//==================================================================================================
//							Beckhoff Automation Poland
//									03.01.2023
//
// Code owner: TG
//
// Sample code to maitenance software limit switches
//
// Used libraries: 
//	Tc2_MC2							|| 3.3.48.0
//	Tc2_System						|| 3.4.26.0
//
//
// 	v2.0 	|| TC v 3.1.4024.35 	|| Second edition - OOP based
// 	v1.0 	|| TC v 3.1.4020.32 	|| First edition
//==================================================================================================
{attribute 'reflection'}
FUNCTION_BLOCK FB_NcSWLimitSwitchCtrlv2
VAR CONSTANT
	udiIDXGRP_OFFS								: UDINT := 16#0000_5000;
END_VAR
VAR
	{attribute 'instance-path'}
	{attribute 'noinit'}
	sInstancePath								: STRING;

	_stRead										: Tc2_MC2.ST_McOutputs;
	_stWrite									: Tc2_MC2.ST_McOutputs;
	_lrLimitSwitchPositionMin					: LREAL 		:= 0;
	_lrLimitSwitchPositionMax					: LREAL 		:= 0;
	_bLimitSwitchStateMin						: BOOL 			:= FALSE;
	_bLimitSwitchStateMax						: BOOL 			:= FALSE;
	bAxisIdError								: BOOL;
END_VAR

PROPERTY LimitSwitchPositionMax 				: LREAL
GET
LimitSwitchPositionMax							:= _lrLimitSwitchPositionMax;
END_GET
SET
_lrLimitSwitchPositionMax						:= LimitSwitchPositionMax;
END_SET
END_PROPERTY

PROPERTY LimitSwitchPositionMin 				: LREAL
GET
LimitSwitchPositionMin							:= _lrLimitSwitchPositionMin;
END_GET
SET
_lrLimitSwitchPositionMin						:= LimitSwitchPositionMin;
END_SET
END_PROPERTY

PROPERTY LimitSwitchStateMax 					: BOOL
GET
LimitSwitchStateMax								:= _bLimitSwitchStateMax;
END_GET
SET
_bLimitSwitchStateMax							:= LimitSwitchStateMax;
END_SET
END_PROPERTY

PROPERTY LimitSwitchStateMin 					: BOOL
GET
LimitSwitchStateMin							:= _bLimitSwitchStateMin;
END_GET
SET
_bLimitSwitchStateMin							:= LimitSwitchStateMin;
END_SET
END_PROPERTY

PROPERTY pRead 							: Tc2_MC2.ST_McOutputs
GET
pRead											:= _stRead;
END_GET
SET
_stRead											:= pRead;
END_SET
END_PROPERTY

PROPERTY pWrite 							: Tc2_MC2.ST_McOutputs
GET
pWrite											:= _stWrite;
END_GET
SET
_stWrite										:= pWrite;
END_SET
END_PROPERTY

// Needs one cycle extra with false execution, after busy false
METHOD ReadBool 								: Tc2_MC2.ST_McOutputs
VAR_INPUT
	bExecute									: BOOL;
	nAxisID										: UDINT;
	nOffset										: UDINT;
END_VAR
VAR_OUTPUT
	bOut										: BOOL;
END_VAR
VAR_INST
	fbADSREAD									: ADSREAD;
	wData										: WORD;
	nStep										: DINT;
END_VAR
VAR
	Out											: Tc2_MC2.ST_McOutputs;
	Message										: STRING;
END_VAR
IF nAxisID = 0 THEN
	
	IF NOT bAxisIdError THEN
		ADSLOGSTR(ADSLOG_MSGTYPE_ERROR,'FB_NcSWLimitSwitchCtrl critical error - Axis ID not assigned! FB instance: %s',sInstancePath);
	END_IF
	
	bAxisIdError 								:= TRUE;
	RETURN;	
END_IF

fbADSREAD(			PORT						:= 500, 
					IDXGRP						:= udiIDXGRP_OFFS + nAxisID, 
					IDXOFFS						:= nOffset, 
					LEN							:= 2, 
					DESTADDR					:= ADR(wData), 
					READ						:= bExecute, 
					BUSY						=> Out.Busy, 
					ERR							=> Out.Error, 
					ERRID						=> Out.ErrorID);

// Fix library issue, one extra cycle + Done
CASE nStep OF
	
	0: 
	
		Out.Error 								:= FALSE;
		Out.ErrorID 							:= 0;

		IF Out.Busy THEN
			nStep								:= nStep + 10;
		END_IF
	
	10:
	
		IF NOT Out.Busy THEN
			Out.Busy							:= TRUE;
			IF Out.Error THEN
				Out.ErrorID						:= 0;
				Out.Error						:= FALSE;
				nStep							:= 1000;
			ELSE
				nStep							:= 100;
			END_IF
		END_IF
		
	100, 1000:

		Out.Done								:= nStep = 100;
		Out.Error								:= nStep = 1000;
		IF Out.Error THEN
			Message := CONCAT('FB_NcSWLimitSwitchCtrl method ReadBool failed - Error ID: ',UDINT_TO_STRING(Out.ErrorID));
			Message := CONCAT(Message, '! FB instance: %s');
			ADSLOGSTR(ADSLOG_MSGTYPE_WARN,Message,sInstancePath);
		END_IF
		
		IF bExecute THEN
			nStep								:= nStep + 1;
		ELSE
			fbADSREAD(	READ					:= FALSE);
			nStep								:= 0;
		END_IF
		
	101, 1001:
	
		Out.Done								:= nStep = 101;
		Out.Error								:= nStep = 1001;
		IF NOT bExecute THEN
			fbADSREAD(	READ					:= FALSE);
			Out.Done							:= FALSE;
			Out.Error							:= FALSE;
			Out.ErrorID							:= 0;
			nStep								:= 0;
		END_IF	

END_CASE

pRead											:= Out;

bOut											:= wData.0;
ReadBool										:= Out;
END_METHOD

METHOD ReadLreal 								: Tc2_MC2.ST_McOutputs
VAR_INPUT
	bExecute									: BOOL;
	nAxisID										: UDINT;
	nOffset										: UDINT;
END_VAR
VAR_OUTPUT
	lrOut										: LREAL;
END_VAR
VAR_INST
	fbADSREAD									: ADSREAD;
	lrData										: LREAL;
	nStep										: DINT;
END_VAR
VAR
	Out											: Tc2_MC2.ST_McOutputs;
	Message										: STRING;
END_VAR
IF nAxisID = 0 THEN
	
	IF NOT bAxisIdError THEN
		ADSLOGSTR(ADSLOG_MSGTYPE_ERROR,'FB_NcSWLimitSwitchCtrl critical error - Axis ID not assigned! FB instance: %s',sInstancePath);
	END_IF
	
	bAxisIdError 								:= TRUE;
	RETURN;	
END_IF

fbADSREAD(			PORT						:= 500, 
					IDXGRP						:= udiIDXGRP_OFFS + nAxisID, 
					IDXOFFS						:= nOffset, 
					LEN							:= 8, 
					DESTADDR					:= ADR(lrData), 
					READ						:= bExecute, 
					BUSY						=> Out.Busy, 
					ERR							=> Out.Error, 
					ERRID						=> Out.ErrorID);

// Fix library issue, one extra cycle + Done
CASE nStep OF
	
	0: 
	
		Out.Error 								:= FALSE;
		Out.ErrorID 							:= 0;

		IF Out.Busy THEN
			nStep								:= nStep + 10;
		END_IF
	
	10:
	
		IF NOT Out.Busy THEN
			Out.Busy							:= TRUE;
			IF Out.Error THEN
				Out.ErrorID						:= 0;
				Out.Error						:= FALSE;
				nStep							:= 1000;
			ELSE
				nStep							:= 100;
			END_IF
		END_IF
		
	100, 1000:

		Out.Done								:= nStep = 100;
		Out.Error								:= nStep = 1000;
		IF Out.Error THEN
			Message := CONCAT('FB_NcSWLimitSwitchCtrl method ReadLreal failed - Error ID: ',UDINT_TO_STRING(Out.ErrorID));
			Message := CONCAT(Message, '! FB instance: %s');
			ADSLOGSTR(ADSLOG_MSGTYPE_WARN,Message,sInstancePath);
		END_IF
		
		IF bExecute THEN
			nStep								:= nStep + 1;
		ELSE
			fbADSREAD(	READ					:= FALSE);
			nStep								:= 0;
		END_IF
		
	101, 1001:
	
		Out.Done								:= nStep = 101;
		Out.Error								:= nStep = 1001;
		IF NOT bExecute THEN
			fbADSREAD(	READ					:= FALSE);
			Out.Done							:= FALSE;
			Out.Error							:= FALSE;
			Out.ErrorID							:= 0;
			nStep								:= 0;
		END_IF	

END_CASE

pRead											:= Out;

lrOut											:= lrData;
ReadLreal										:= Out;
END_METHOD

METHOD ReadParams 								: Tc2_MC2.ST_McOutputs
VAR_INPUT
	bExecute									: BOOL;
	nAxisID										: UDINT;
END_VAR
VAR_INST
	stOut	 									: Tc2_MC2.ST_McOutputs;
	nStep										: DINT;
END_VAR
VAR
	Out	 										: Tc2_MC2.ST_McOutputs;
END_VAR
CASE nStep OF

	0: 
		IF bExecute THEN
			stOut.Busy							:= TRUE;
			nStep								:= nStep + 5;
		END_IF
		
	5:

		Out 									:= ReadValueMin(bExecute := TRUE, nAxisID := nAxisID);
		IF Out.Busy THEN
			nStep								:= nStep + 5;
		END_IF
	
	10:
	
		Out 									:= ReadValueMin(bExecute := FALSE, nAxisID := nAxisID);
		IF Out.Done THEN
			nStep								:= nStep + 5;
		ELSIF Out.Error THEN
			nStep								:= 1000;
		END_IF
	
	15: 
	
		Out 									:= ReadValueMax(bExecute := TRUE, nAxisID := nAxisID);
		IF Out.Busy THEN
			nStep								:= nStep + 5;
		END_IF
		
	20:
	
		Out 									:= ReadValueMax(bExecute := FALSE, nAxisID := nAxisID);
		IF Out.Done THEN
			nStep								:= nStep + 5;
		ELSIF Out.Error THEN
			nStep								:= 1000;
		END_IF
	
	25: 
	
		Out 									:= ReadStateMin(bExecute := TRUE, nAxisID := nAxisID);
		IF Out.Busy THEN
			nStep								:= nStep + 5;
		END_IF
		
	30:
	
		Out 									:= ReadStateMin(bExecute := FALSE, nAxisID := nAxisID);
		IF Out.Done THEN
			nStep								:= nStep + 5;
		ELSIF Out.Error THEN
			nStep								:= 1000;
		END_IF
	
	35: 
	
		Out 									:= ReadStateMax(bExecute := TRUE, nAxisID := nAxisID);
		IF Out.Busy THEN
			nStep								:= nStep + 5;
		END_IF
		
	40:
	
		Out 									:= ReadStateMax(bExecute := FALSE, nAxisID := nAxisID);
		IF Out.Done THEN
			nStep								:= 100;
		ELSIF Out.Error THEN
			nStep								:= 1000;
		END_IF
		
	100, 1000:

		stOut.Busy								:= FALSE;
		stOut.Done								:= nStep = 100;
		stOut.Error								:= nStep = 1000;
		nStep									:= nStep + 1;
		
	101, 1001:
	
		IF NOT bExecute THEN
			stOut.Busy							:= FALSE;
			stOut.Done							:= FALSE;
			stOut.Error							:= FALSE;
			nStep								:= 0;			
		END_IF

END_CASE

ReadParams										:= stOut;
END_METHOD

METHOD ReadStateMax 							: Tc2_MC2.ST_McOutputs
VAR_INPUT
	bExecute									: BOOL;
	nAxisID										: UDINT;
END_VAR
VAR
	bOut										: BOOL;
END_VAR
ReadStateMax 									:= ReadBool(	bExecute 	:= bExecute, 
																nAxisID 	:= nAxisID, 
																nOffset 	:= 16#0000_000C, 
																bOut 		=> bOut);

LimitSwitchStateMax								:= bOut;
END_METHOD

METHOD ReadStateMin 							: Tc2_MC2.ST_McOutputs
VAR_INPUT
	bExecute									: BOOL;
	nAxisID										: UDINT;
END_VAR
VAR
	bOut										: BOOL;
END_VAR
ReadStateMin 									:= ReadBool(	bExecute 	:= bExecute, 
																nAxisID 	:= nAxisID, 
																nOffset 	:= 16#0000_000B, 
																bOut 		=> bOut);
																
LimitSwitchStateMin								:= bOut;
END_METHOD

METHOD ReadValueMax 							: Tc2_MC2.ST_McOutputs
VAR_INPUT
	bExecute									: BOOL;
	nAxisID										: UDINT;
END_VAR
VAR
	lrOut										: LREAL;
END_VAR
ReadValueMax 									:= ReadLreal(	bExecute 	:= bExecute, 
																nAxisID 	:= nAxisID, 
																nOffset 	:= 16#0000_000E, 
																lrOut 		=> lrOut);
																
LimitSwitchPositionMax							:= lrOut;
END_METHOD

METHOD ReadValueMin 							: Tc2_MC2.ST_McOutputs
VAR_INPUT
	bExecute									: BOOL;
	nAxisID										: UDINT;
END_VAR
VAR
	lrOut										: LREAL;
END_VAR
ReadValueMin 									:= ReadLreal(	bExecute 	:= bExecute, 
																nAxisID 	:= nAxisID, 
																nOffset 	:= 16#0000_000D, 
																lrOut 		=> lrOut);
																
LimitSwitchPositionMin							:= lrOut;
END_METHOD

METHOD WriteBool 								: Tc2_MC2.ST_McOutputs
VAR_INPUT
	bExecute									: BOOL;
	bValue										: BOOL;
	nAxisID										: UDINT;
	nOffset										: UDINT;
END_VAR
VAR_INST
	fbADSWRITE									: ADSWRITE;
	wData										: WORD;
	nStep										: DINT;
END_VAR
VAR
	Out											: Tc2_MC2.ST_McOutputs;
	Message										: STRING;
END_VAR
IF nAxisID = 0 THEN
	
	IF NOT bAxisIdError THEN
		ADSLOGSTR(ADSLOG_MSGTYPE_ERROR,'FB_NcSWLimitSwitchCtrl critical error - Axis ID not assigned! FB instance: %s',sInstancePath);
	END_IF
	
	bAxisIdError 								:= TRUE;
	RETURN;	
END_IF

wData.0 										:= bValue;

fbADSWRITE(			PORT						:= 500, 
					IDXGRP						:= udiIDXGRP_OFFS + nAxisID, 
					IDXOFFS						:= nOffset, 
					LEN							:= 2, 
					SRCADDR						:= ADR(wData), 
					WRITE						:= bExecute, 
					BUSY						=> Out.Busy, 
					ERR							=> Out.Error, 
					ERRID						=> Out.ErrorID);

// Fix library issue, one extra cycle + Done
CASE nStep OF
	
	0: 
	
		Out.Error 								:= FALSE;
		Out.ErrorID 							:= 0;

		IF Out.Busy THEN
			nStep								:= nStep + 10;
		END_IF
	
	10:
	
		IF NOT Out.Busy THEN
			Out.Busy							:= TRUE;
			IF Out.Error THEN
				Out.ErrorID						:= 0;
				Out.Error						:= FALSE;
				nStep							:= 1000;
			ELSE
				nStep							:= 100;
			END_IF
		END_IF
		
	100, 1000:

		Out.Done								:= nStep = 100;
		Out.Error								:= nStep = 1000;
		IF Out.Error THEN
			Message := CONCAT('FB_NcSWLimitSwitchCtrl method WriteBool failed - Error ID: ',UDINT_TO_STRING(Out.ErrorID));
			Message := CONCAT(Message, '! FB instance: %s');
			ADSLOGSTR(ADSLOG_MSGTYPE_WARN,Message,sInstancePath);
		END_IF
		
		IF bExecute THEN
			nStep								:= nStep + 1;
		ELSE
			fbADSWRITE(	WRITE					:= FALSE);
			nStep								:= 0;
		END_IF
		
	101, 1001:
	
		Out.Done								:= nStep = 101;
		Out.Error								:= nStep = 1001;
		IF NOT bExecute THEN
			fbADSWRITE(	WRITE					:= FALSE);
			Out.Done							:= FALSE;
			Out.Error							:= FALSE;
			Out.ErrorID							:= 0;
			nStep								:= 0;
		END_IF	

END_CASE

pWrite											:= Out;
WriteBool										:= Out;
END_METHOD

METHOD WriteLreal 								: Tc2_MC2.ST_McOutputs
VAR_INPUT
	bExecute									: BOOL;
	lrValue										: LREAL;
	nAxisID										: UDINT;
	nOffset										: UDINT;
END_VAR
VAR_INST
	fbADSWRITE									: ADSWRITE;
	nStep										: DINT;
END_VAR
VAR
	Out											: Tc2_MC2.ST_McOutputs;
	Message										: STRING;
END_VAR
IF nAxisID = 0 THEN
	
	IF NOT bAxisIdError THEN
		ADSLOGSTR(ADSLOG_MSGTYPE_ERROR,'FB_NcSWLimitSwitchCtrl critical error - Axis ID not assigned! FB instance: %s',sInstancePath);
	END_IF
	
	bAxisIdError 								:= TRUE;
	RETURN;	
END_IF

fbADSWRITE(			PORT						:= 500, 
					IDXGRP						:= udiIDXGRP_OFFS + nAxisID, 
					IDXOFFS						:= nOffset, 
					LEN							:= 8, 
					SRCADDR						:= ADR(lrValue), 
					WRITE						:= bExecute, 
					BUSY						=> Out.Busy, 
					ERR							=> Out.Error, 
					ERRID						=> Out.ErrorID);

// Fix library issue, one extra cycle + Done
CASE nStep OF
	
	0: 
	
		Out.Error 								:= FALSE;
		Out.ErrorID 							:= 0;

		IF Out.Busy THEN
			nStep								:= nStep + 10;
		END_IF
	
	10:
	
		IF NOT Out.Busy THEN
			Out.Busy							:= TRUE;
			IF Out.Error THEN
				Out.ErrorID						:= 0;
				Out.Error						:= FALSE;
				nStep							:= 1000;
			ELSE
				nStep							:= 100;
			END_IF
		END_IF
		
	100, 1000:

		Out.Done								:= nStep = 100;
		Out.Error								:= nStep = 1000;
		IF Out.Error THEN
			Message := CONCAT('FB_NcSWLimitSwitchCtrl method WriteLreal failed - Error ID: ',UDINT_TO_STRING(Out.ErrorID));
			Message := CONCAT(Message, '! FB instance: %s');
			ADSLOGSTR(ADSLOG_MSGTYPE_WARN,Message,sInstancePath);
		END_IF
		
		IF bExecute THEN
			nStep								:= nStep + 1;
		ELSE
			fbADSWRITE(	WRITE					:= FALSE);
			nStep								:= 0;
		END_IF
		
	101, 1001:
	
		Out.Done								:= nStep = 101;
		Out.Error								:= nStep = 1001;
		IF NOT bExecute THEN
			fbADSWRITE(	WRITE					:= FALSE);
			Out.Done							:= FALSE;
			Out.Error							:= FALSE;
			Out.ErrorID							:= 0;
			nStep								:= 0;
		END_IF	

END_CASE

pWrite											:= Out;
WriteLreal										:= Out;
END_METHOD

METHOD WriteParams 								: Tc2_MC2.ST_McOutputs
VAR_INPUT
	bExecute									: BOOL;
	nAxisID										: UDINT;
END_VAR
VAR_INST
	stOut	 									: Tc2_MC2.ST_McOutputs;
	nStep										: DINT;
	lrLimitSwitchPositionMin					: LREAL 		:= 0;
	lrLimitSwitchPositionMax					: LREAL 		:= 0;
	bLimitSwitchStateMin						: BOOL 			:= FALSE;
	bLimitSwitchStateMax						: BOOL 			:= FALSE;
END_VAR
VAR
	Out	 										: Tc2_MC2.ST_McOutputs;
END_VAR
CASE nStep OF

	0: 
		IF bExecute THEN
			lrLimitSwitchPositionMin			:= LimitSwitchPositionMin;
			lrLimitSwitchPositionMax			:= LimitSwitchPositionMax;
			bLimitSwitchStateMin				:= LimitSwitchStateMin;
			bLimitSwitchStateMax				:= LimitSwitchStateMax;
			stOut.Busy							:= TRUE;
			nStep								:= nStep + 5;
		END_IF
		
	5:

		LimitSwitchPositionMin					:= lrLimitSwitchPositionMin;
		Out 									:= WriteValueMin(bExecute := TRUE, nAxisID := nAxisID);
		IF Out.Busy THEN
			nStep								:= nStep + 5;
		END_IF
	
	10:
	
		Out 									:= WriteValueMin(bExecute := FALSE, nAxisID := nAxisID);
		IF Out.Done THEN
			nStep								:= nStep + 5;
		ELSIF Out.Error THEN
			nStep								:= 1000;
		END_IF
	
	15: 
	
		LimitSwitchPositionMax					:= lrLimitSwitchPositionMax;
		Out 									:= WriteValueMax(bExecute := TRUE, nAxisID := nAxisID);
		IF Out.Busy THEN
			nStep								:= nStep + 5;
		END_IF
		
	20:
	
		Out 									:= WriteValueMax(bExecute := FALSE, nAxisID := nAxisID);
		IF Out.Done THEN
			nStep								:= nStep + 5;
		ELSIF Out.Error THEN
			nStep								:= 1000;
		END_IF
	
	25: 
	
		LimitSwitchStateMin						:= bLimitSwitchStateMin;
		Out 									:= WriteStateMin(bExecute := TRUE, nAxisID := nAxisID);
		IF Out.Busy THEN
			nStep								:= nStep + 5;
		END_IF
		
	30:
	
		Out 									:= WriteStateMin(bExecute := FALSE, nAxisID := nAxisID);
		IF Out.Done THEN
			nStep								:= nStep + 5;
		ELSIF Out.Error THEN
			nStep								:= 1000;
		END_IF
	
	35: 

		LimitSwitchStateMax						:= bLimitSwitchStateMax;	
		Out 									:= WriteStateMax(bExecute := TRUE, nAxisID := nAxisID);
		IF Out.Busy THEN
			nStep								:= nStep + 5;
		END_IF
		
	40:
	
		Out 									:= WriteStateMax(bExecute := FALSE, nAxisID := nAxisID);
		IF Out.Done THEN
			nStep								:= 100;
		ELSIF Out.Error THEN
			nStep								:= 1000;
		END_IF
		
	100, 1000:

		stOut.Busy								:= FALSE;
		stOut.Done								:= nStep = 100;
		stOut.Error								:= nStep = 1000;
		nStep									:= nStep + 1;
		
	101, 1001:
	
		IF NOT bExecute THEN
			stOut.Busy							:= FALSE;
			stOut.Done							:= FALSE;
			stOut.Error							:= FALSE;
			nStep								:= 0;			
		END_IF

END_CASE

WriteParams										:= stOut;
END_METHOD

METHOD WriteStateMax 							: Tc2_MC2.ST_McOutputs
VAR_INPUT
	bExecute									: BOOL;
	nAxisID										: UDINT;
END_VAR
WriteStateMax 									:= WriteBool(	bExecute 	:= bExecute,
 																bValue		:= LimitSwitchStateMax,
																nAxisID 	:= nAxisID, 
																nOffset 	:= 16#0000_000C);
END_METHOD

METHOD WriteStateMin 							: Tc2_MC2.ST_McOutputs
VAR_INPUT
	bExecute									: BOOL;
	nAxisID										: UDINT;
END_VAR
WriteStateMin 									:= WriteBool(	bExecute 	:= bExecute,
 																bValue		:= LimitSwitchStateMin,
																nAxisID 	:= nAxisID, 
																nOffset 	:= 16#0000_000B);
END_METHOD

METHOD WriteValueMax 							: Tc2_MC2.ST_McOutputs
VAR_INPUT
	bExecute									: BOOL;
	nAxisID										: UDINT;
END_VAR
WriteValueMax 									:= WriteLreal(	bExecute 	:= bExecute, 
																lrValue		:= LimitSwitchPositionMax,
																nAxisID 	:= nAxisID, 
																nOffset 	:= 16#0000_000E);
END_METHOD

METHOD WriteValueMin 							: Tc2_MC2.ST_McOutputs
VAR_INPUT
	bExecute									: BOOL;
	nAxisID										: UDINT;
END_VAR
WriteValueMin 									:=  WriteLreal(	bExecute 	:= bExecute, 
																lrValue		:= LimitSwitchPositionMin,
																nAxisID 	:= nAxisID, 
																nOffset 	:= 16#0000_000D);
END_METHOD

END_FUNCTION_BLOCK

(* stored: Version 1.2.0.0, ProductVersion 3.1.4026.13, FileIdentifier ae219ea2d2b0024689205b88a104a1f517b1b33b, FileSignature 88410e2c15fa21e1e8e032fbdb6d5dc5a199472570b3a6efb8508ba3581f4ead063faf0ef7722242d1407dc7b5ddacc6b1a5477e9f049a4e1c8ecc99e81a0024f0f04d9da76b04f8d3e97401dcde742c45c4ec9001483baab24f568a3ff70afb8320df6158359617633ff5d515d6e93e5f9258b5c293e1938ccae2259e9e8d515e329996f6cd16287ff7d2c5e6fb423f3bc268029f4c0945ef48819fb34957c5145906f532d8f6fd05557712a21f7d111d8ec6a011f5ea31f79d66dc4f4841cba3d8e8ae5ebe65811bbfdc79bdf6e32f7c507d3ac1e9e669b7a504926958363392a7b6d3ce94931f48e42550dc13a10b77fa56a7070e63e21d77a06a622cefac
   POU FB_NcSWLimitSwitchCtrlv2: Id {f1ad3452-a250-4d9d-983c-dd0efabdf0d1}, SpecialFunc None
   Folder General: Id {3107b5a0-2e6d-409a-a45d-2a85b08105ad}
   Folder Properties: Id {d3a7f47e-52ec-45aa-b773-85d632f8f1fa}
   Folder Special: Id {278e8b73-9fe4-41da-9046-2d5fd92a3174}
   Folder Sum: Id {f490a69d-3e01-4c5a-a516-f430f22e2a03}
   Property LimitSwitchPositionMax: Id {88e41b6e-b0f3-46e7-8966-ba50d9ac1155}
   Get Get: Id {e81ec829-2576-4559-b466-97a590dba28e}
   Set Set: Id {3c968c53-3e17-4ac3-aea1-f450a8de937e}
   Property LimitSwitchPositionMin: Id {ee073076-01c4-4f8a-b44d-443c5ab5f143}
   Get Get: Id {27786fb6-bb4d-4252-9b80-33d2a722078b}
   Set Set: Id {1e7f97ee-7609-42c5-9cfb-f6ee562361ac}
   Property LimitSwitchStateMax: Id {4779f2f8-9464-425d-be43-df77c9b9af85}
   Get Get: Id {343de313-6176-44fe-96ce-42afdc1f34a3}
   Set Set: Id {a4e4e87a-1c16-43fe-8152-9b1fc8adfc58}
   Property LimitSwitchStateMin: Id {41a9026c-4e2f-462c-9240-d8ccaf494d71}
   Get Get: Id {8d4b1210-4fac-4dad-848c-ed38a12555c8}
   Set Set: Id {13a0a108-a23d-4e73-8f49-0874b85f7049}
   Property pRead: Id {2419c57b-ae9d-4a27-96c8-06d5d95daaba}
   Get Get: Id {c5b06164-c0a1-48ec-a7c8-a6d96cfa6430}
   Set Set: Id {6135818c-574c-4c95-b836-afef7d85d93e}
   Property pWrite: Id {e1646478-07d7-4735-8adf-e051b2c6d85b}
   Get Get: Id {0707df5f-4283-4c92-844d-b4cd6588081e}
   Set Set: Id {e5b1be28-5af6-45ab-849b-b5755b030e05}
   Method ReadBool: Id {da5a20eb-b604-4064-bfb6-61ecfb6c034e}
   Method ReadLreal: Id {f8267c7d-d392-4bfd-bccb-a5a767a9bc4b}
   Method ReadParams: Id {dfdb63e0-67be-4d77-a7b7-b72404cd84ba}
   Method ReadStateMax: Id {6c5c4858-0555-49d8-a82f-36dc8ae7db41}
   Method ReadStateMin: Id {389af012-88a6-4e73-abf0-0e3924805f5b}
   Method ReadValueMax: Id {52157751-0a96-48a3-9e11-dd1cdd73c3d7}
   Method ReadValueMin: Id {f74951ef-c5e7-4ef1-a590-bb3efd098dca}
   Method WriteBool: Id {0f86a79d-26bb-4725-844c-bc11333929da}
   Method WriteLreal: Id {69d5dfb5-6a12-4355-b1ab-ed172b302642}
   Method WriteParams: Id {b525ad41-16de-4e48-96ba-140bb7ae6a53}
   Method WriteStateMax: Id {be7fda39-bb34-4bf2-9738-6c4d78ecd450}
   Method WriteStateMin: Id {bf4cb29c-dadb-469c-84f8-0c16f3654c39}
   Method WriteValueMax: Id {1fe1bbad-9fcf-4b2f-a52a-53188895ed7e}
   Method WriteValueMin: Id {a6b2e1ef-f7ac-41a2-8b72-6c49a0244356} *)
